PROGRAM PTC_RX_COM
VAR
	send_message : PTC_Send_Message;
	receive_messages : PTC_Receive_Messages;
	LV_BAT_Par : FB_CAN_LV;
END_VAR

receive_messages(CAN_OUTPUTS := GVL_PT.CAN_OUTPUTS, CAN_INPUTS := GVL_PT.CAN_INPUTS);
LV_BAT_Par();

END_PROGRAM

(* stored: Version 1.1.0.1
   POU PTC_RX_COM: Id {4d778e1c-c04b-4095-bcb6-a923efd7ffab}, SpecialFunc None *)
